{attribute 'linkalways'} 
{attribute 'no_explicit_call' := 'This FB is a CLASS and must be accessed using methods or properties'}
{attribute 'enable_dynamic_creation'}
FUNCTION_BLOCK FINAL SEL_USINT EXTENDS Node
VAR
	g : _BOOL(FALSE);
	in1 : _USINT(0);
	in2 : _USINT(0);
	out : _USINT(0);
END_VAR

METHOD PUBLIC Clone : I_Node
VAR
	pNode : POINTER TO SEL_USINT;
END_VAR
pNode := __NEW(SEL_USINT);
Clone := pNode^;
END_METHOD

METHOD FB_init : BOOL
VAR_INPUT
	bInitRetains : BOOL; // if TRUE, the retain variables are initialized (warm start / cold start)
	bInCopyCode : BOOL;  // if TRUE, the instance afterwards gets moved into the copy code (online change)
END_VAR
AddInput('g',THIS^.g);
AddInput('in1',THIS^.in1);
AddInput('in2',THIS^.in2);
AddOutput('out', THIS^.out);
END_METHOD

METHOD PROTECTED OnExecute
VAR
END_VAR
IF g.value THEN
	out.value := in2.value;
ELSE
	out.value := in1.value;
END_IF
END_METHOD

END_FUNCTION_BLOCK

(* stored: Version 1.1.0.1, ProductVersion 3.1.4024.15
   POU SEL_USINT: Id {f185fb63-3edc-44ee-905c-f8db2b07611f}, SpecialFunc None
   Folder Constructor: Id {40643acf-18c2-48e6-8709-068e9c4a985b}
   Method Clone: Id {565b2bfd-bada-40f7-9153-c5beb5cd0108}
   Method FB_init: Id {bf43c16a-7d0b-4016-92e1-561092a52d16}
   Method OnExecute: Id {3bb5ecc2-93c6-428a-90d6-ef3789062489} *)
